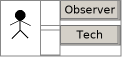
VISUALIZATION VISU_OperatorStatus_Old  // 122x57
VAR_IN_OUT
	status : OperatorStatus;
	process : ChangeOperatorStateProcess;
END_VAR
    Frame (40,0 20x30)
        shows VISU_State_gray_green(state := status.observer)
    Button (60,0 60x20), "Observer", input disabled if: process.statuses.enabledStatus.disabled
        OnMouseClick: execute { process.set.state := OperatorStates.OBSERVER; process.do_request := TRUE; }
        OnMouseDown: execute {  }
    Button (60,25 60x20), "Tech", input disabled if: process.statuses.enabledStatus.disabled
        OnMouseClick: execute { process.set.state := OperatorStates.TECH; process.do_request := TRUE; }
        OnMouseDown: execute {  }
    Frame (40,25 20x30)
        shows VISU_State_gray_orange(state := status.tech)
    Line (20,30) (20,20)
    Line (12,38) (20,30)
    Line (28,38) (20,30)
    Line (20,20) (10,25)
    Line (20,20) (30,25)
    Ellipse (15,10 10x10)
END_VISUALIZATION

(* stored: Version 1.1.0.1, ProductVersion 3.1.4019.2
   Visu VISU_OperatorStatus_Old: Id {627fae61-9327-4837-86c3-60703dfa7889} *)
